(* IEC 61131-3 sources: AXOpen/src/_components.cognex.vision/ctrl/src/AxoInsight/v_6_0_0/TypeStructuresAndEnums, 2 files *)

(* ---- AxoInsight_AcquisitionStatus.st ---- *)
NAMESPACE AXOpen.Components.Cognex.Vision.v_6_0_0_0
    TYPE
        {#ix-attr:[Container(Layout.Wrap)]}
        {S7.extern=ReadWrite}
        AxoInsight_AcquisitionStatus :
        STRUCT
            {#ix-set:AttributeName = "<#Trigger ready#>"}
            TriggerReady 		:	BOOL;
            {#ix-set:AttributeName = "<#Trigger acknowledge#>"}
            TriggerAcknowledge 	:	BOOL;
            {#ix-set:AttributeName = "<#Exposure complete#>"}
            ExposureComplete	:	BOOL;
            {#ix-set:AttributeName = "<#Missed acquisition#>"}
            MissedAcquisition 	:	BOOL;
            {#ix-set:AttributeName = "<#Offline reason 0#>"}
            OfflineReason0      :   BOOL;
            {#ix-set:AttributeName = "<#Offline reason 1#>"}
            OfflineReason1      :   BOOL;
            {#ix-set:AttributeName = "<#Offline reason 2#>"}
            OfflineReason2      :   BOOL;
            {#ix-set:AttributeName = "<#Online#>"}
            Online              :   BOOL;
            {#ix-set:AttributeName = "<#Acquisition ID#>"}
            AcquisitionID       :   UINT;
        END_STRUCT;
    END_TYPE
END_NAMESPACE

(* ---- AxoInsight_Status.st ---- *)
USING AXOpen.Core;
NAMESPACE AXOpen.Components.Cognex.Vision.v_6_0_0_0
    {#ix-attr:[Container(Layout.Stack)]}
    {S7.extern=ReadWrite}
    CLASS AxoInsight_Status EXTENDS AXOpen.Components.Abstractions.AxoComponent_Status
        VAR PUBLIC
            {#ix-attr:[Container(Layout.Wrap)]}
            {#ix-set:AttributeName = "<#Current job name#>"}
            CurrentJobName : STRING;
            {#ix-set:AttributeName = "<#Current job number#>"}
            CurrentJobNumber : UINT;
            {#ix-set:AttributeName = "<#Result data size#>"}
            ResultDataSize : eAxoInsight_ResultDataSize := eAxoInsight_ResultDataSize#RESULT_DATA_SIZE_INVALID;
            {#ix-set:AttributeName = "<#User data size#>"}
            UserDataSize : eAxoInsight_UserDataSize := eAxoInsight_UserDataSize#USER_DATA_SIZE_INVALID;
        END_VAR
    END_CLASS
END_NAMESPACE
